TYPE ST_CRC_Params :
STRUCT
    bitWidth      		: BYTE;
    polynomial       	: XWORD;
    initCRC       		: XWORD;
    reflectInitial      : BOOL;
    reflected     		: BOOL;
    xorOut     			: XWORD;
    check      			: XWORD;
    residue    			: XWORD;
END_STRUCT
END_TYPE

(* stored: Version 1.1.0.1
   DUT ST_CRC_Params: Id {edd7a7fb-6b87-408c-b98a-341884341885} *)
